KUKA KRL program: BrakeTestPark.src, BrakeTestPark.dat

--- BrakeTestPark.src ---
&ACCESS RV
&REL 1
&COMMENT parkposition
&PARAM EDITMASK = *
&PARAM TEMPLATE = C:\KRC\Roboter\Template\vorgabe
&PARAM DISKPATH = KRC:\R1\TP\BrakeTest
DEF BrakeTestPark( )
;FOLD INI
  ;FOLD BASISTECH INI
    GLOBAL INTERRUPT DECL 3 WHEN $STOPMESS==TRUE DO IR_STOPM ( )
    INTERRUPT ON 3
  ;ENDFOLD (BASISTECH INI)
  ;FOLD USER INI
    ;Make your modifications here
  ;ENDFOLD (USER INI)
;ENDFOLD (INI)
;Teach here the motion to the parking position. The parking position is needed when the robot has failed the brake test.
;FOLD {h}
WHILE ParkPositionInNotValid()
  MsgDialog(SUCCESS,"ParkPositionIsNotValid",brakeTestMdbName[],,,,,,,"Ok")
  HALT
ENDWHILE
;ENDFOLD
;FOLD SPTP ParkPosition Vel=10 % DEFAULT Tool[1] Base[0] ;%{PE}
;FOLD Parameters ;%{h}
;Params IlfProvider=kukaroboter.basistech.inlineforms.movement.spline; Kuka.IsGlobalPoint=False; Kuka.PointName=ParkPosition; Kuka.BlendingEnabled=False; Kuka.MoveDataPtpName=DEFAULT; Kuka.VelocityPtp=10; Kuka.VelocityFieldEnabled=True; Kuka.ColDetectFieldEnabled=True; Kuka.CurrentCDSetIndex=0; Kuka.MovementParameterFieldEnabled=True; IlfCommand=SPTP
;ENDFOLD
SPTP XParkPosition WITH $VEL_AXIS[1] = SVEL_JOINT(10.0), $TOOL = STOOL2(FParkPosition), $BASE = SBASE(FParkPosition.BASE_NO), $IPO_MODE = SIPO_MODE(FParkPosition.IPO_FRAME), $LOAD = SLOAD(FParkPosition.TOOL_NO), $ACC_AXIS[1] = SACC_JOINT(PDEFAULT), $APO = SAPO_PTP(PDEFAULT), $GEAR_JERK[1] = SGEAR_JERK(PDEFAULT), $COLLMON_TOL_PRO[1] = USE_CM_PRO_VALUES(0)
;ENDFOLD
END
;FOLD {h}
Global DEFFCT BOOL ParkPositionInNotValid()
RETURN ((XParkPosition.A1 == 999) AND (XParkPosition.A2 == 999) AND (XParkPosition.A3 == 999) AND (XParkPosition.A4 == 999) AND (XParkPosition.A5 == 999) AND (XParkPosition.A6 == 999) AND (XParkPosition.E1 == 999) AND (XParkPosition.E2 == 999) AND (XParkPosition.E3 == 999) AND (XParkPosition.E4 == 999) AND (XParkPosition.E5 == 999) AND (XParkPosition.E6 == 999))
ENDFCT
;ENDFOLD

--- BrakeTestPark.dat ---
&ACCESS RV
&REL 1
&COMMENT parkposition
&PARAM EDITMASK = *
&PARAM TEMPLATE = C:\KRC\Roboter\Template\vorgabe
&PARAM DISKPATH = KRC:\R1\TP\BrakeTest
DEFDAT  BRAKETESTPARK PUBLIC
;FOLD EXTERNAL DECLARATIONS;%{PE}%MKUKATPBASIS,%CEXT,%VCOMMON,%P
;FOLD BASISTECH EXT;%{PE}%MKUKATPBASIS,%CEXT,%VEXT,%P
EXT  BAS (BAS_COMMAND  :IN,REAL  :IN )
DECL INT SUCCESS
;ENDFOLD (BASISTECH EXT)
;FOLD USER EXT;%{E}%MKUKATPUSER,%CEXT,%VEXT,%P
;Make here your modifications
;ENDFOLD (USER EXT)
;ENDFOLD (EXTERNAL DECLERATIONS)
DECL E6AXIS XParkPosition={A1 999.000,A2 999.000,A3 999.000,A4 999.000,A5 999.000,A6 999.000,E1 999.000,E2 999.000,E3 999.000,E4 999.000,E5 999.000,E6 999.000}
DECL FDAT FParkPosition={TOOL_NO 1,BASE_NO 0,IPO_FRAME #BASE,POINT2[] " "}
ENDDAT
